FUNCTION_BLOCK FB_PS_Grid EXTENDS FB_PS
VAR_INPUT
END_VAR
VAR_OUTPUT
END_VAR
VAR
  sCG : ARRAY[1..iCPr_NB_PH_PS_MAX] OF I_Correction_Grid;
  
  nRowMap : ARRAY[1..iCPr_NB_PH_PS_MAX,1..2] OF DINT; (*PH[x, [min, max]] Min..Max ROI row per head*)
  sDefGridSettings : ST_DefGridSettings;
END_VAR

METHOD newGridPoint : BOOL
VAR_INPUT
  sPoint : ST_DeformationPointAccurate;
END_VAR
VAR
  bOK : BOOL;
  bLimited : BOOL;
  i : UDINT;
  sPointPx : ST_DeformationPoint;
END_VAR
// write to head(s)
FOR i:=1 TO nPh DO
  
  //Check if point in scope of printhead (rows) (NOTE: could be remo)
  IF sPoint.row >= nRowMap[i,1] AND sPoint.row <= nRowMap[i,2] THEN

    // write DefGrid point
    sPointPx := F_EncodeDeformationPoint(sPoint:=sPoint, nResolution:=1);   // convert point to fixed point (floor)
    bOK := sCG[i].writeCorrectionPoint(sPoint:=sPointPx);
    IF NOT bOK THEN 
      LogWarning(F_Concat6('Could not write GridPoint to PH[', TO_STRING(i), '] c:', TO_STRING(sPoint.col), '/r:', TO_STRING(sPoint.row)));
    END_IF
	END_IF
END_FOR

newGridPoint := TRUE;
END_METHOD

METHOD printPrepare
VAR
  i : UDINT;
END_VAR
// set print enable 
FOR i:=1 TO nPh DO
  sPh[i].setPrintEnable(bPrintEnable := sPh[i].bEnable AND _bPrintEnable);  // if ph is enabled and ps print enable is set
END_FOR
END_METHOD

METHOD registerCG : BOOL
VAR_INPUT
      iNewPh : I_PH;                // printhead interface
      iNewCG : I_Correction_Grid;   // correction grid interface
END_VAR
IF iNewCG = 0 OR iNewCG = 0 THEN LogError('registerCG: Invalid parameter'); F_Report_Error(ErrType:=EN_REPORT_ERROR_TYPE.Report_Error_0Pointer); RETURN; END_IF
IF THIS^.registerPh(iNewPh:=iNewPh) THEN
    sCG[nPh] := iNewCG; //add CG same as printhead, they are in sync
END_IF
END_METHOD

METHOD setGrid
VAR_INPUT
  sGrid : ST_DefGridSettings;
END_VAR
VAR
  i : UDINT;
END_VAR
// grid settings checks
IF sGrid.nGridPitchX = 0 OR sGrid.nGridPitchY = 0 OR sGrid.nGridPoints = 0 THEN
  LogError('Invalid grid settings');
  RETURN;
END_IF

// save grid settings
sDefGridSettings :=sGrid;

// set grid on PH 
FOR i:=1 TO nPh DO
  sCG[i].setGrid(sGrid:=sGrid);
  
  (* setup grid filter in PS (for better performance, pre-filter points before sending to ph) 
      this could removed so we have the RIO calculation only once.*)
  IF sPh[i] <> 0 AND sCG[i] <> 0 THEN
    // lower row bound
    nRowMap[i,1]:=sPh[i].nPositionY / UDINT_TO_DINT(sDefGridSettings.nGridPitchY);   // floor
    // upper row bound
    nRowMap[i,2]:=(sPh[i].nPositionY + sPh[i].nHeadWidth) / UDINT_TO_DINT(sDefGridSettings.nGridPitchY) + 1;
    {warning 'TODO: review with RIO calculation if FPGA is right'}
    nRowMap[i,2]:=nRowMap[i,1] + GVL_Deformation.nC_GridRoiRows - 1;
    
    // limit to grid scope
    nRowMap[i,1] := LIMIT(0,nRowMap[i,1],UDINT_TO_DINT(sDefGridSettings.nGridSizeY));
    nRowMap[i,2] := LIMIT(0,nRowMap[i,2],UDINT_TO_DINT(sDefGridSettings.nGridSizeY));
  ELSE
    F_Report_Error(ErrType:=EN_REPORT_ERROR_TYPE.Report_Error_0Pointer);
  END_IF  
END_FOR
END_METHOD

END_FUNCTION_BLOCK

(* stored: Version 1.1.0.1, ProductVersion 3.1.4024.3
   POU FB_PS_Grid: Id {9c5e3abb-c4bc-4a7b-938e-25a9d7e81622}, SpecialFunc None
   Method newGridPoint: Id {9f9665fc-9dda-4195-aa07-7605112b126e}
   Method printPrepare: Id {fdf28f07-247a-4033-92d5-ffed501251f9}
   Method registerCG: Id {15a4429f-45fa-4f57-9655-f7ccd96f089d}
   Method setGrid: Id {5a0bdc95-65ff-4d0e-972d-23940539c977} *)
